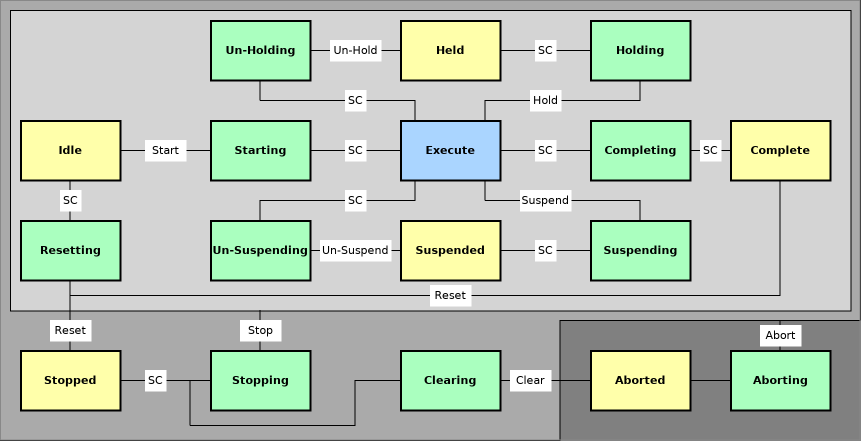
VISUALIZATION VFM_PackML  // 861x441
VAR_IN_OUT
	HMI : ST_PackMLBaseModule_HMI;
END_VAR
    Rectangle (560,320 301x121)
    Rectangle (10,10 841x301)
    Rectangle (590,350 101x61), "Aborted", colour toggle: HMI.Status.State = Tc3_PackML_V2.E_PMLState.ePMLState_Aborted
    Rectangle (400,350 101x61), "Clearing", colour toggle: HMI.Status.State = Tc3_PackML_V2.E_PMLState.ePMLState_Clearing
    Rectangle (210,350 101x61), "Stopping", colour toggle: HMI.Status.State = Tc3_PackML_V2.E_PMLState.ePMLState_Stopping
    Rectangle (20,350 101x61), "Stopped", colour toggle: HMI.Status.State = Tc3_PackML_V2.E_PMLState.ePMLState_Stopped
    Rectangle (20,220 101x61), "Resetting", colour toggle: HMI.Status.State = Tc3_PackML_V2.E_PMLState.ePMLState_Resetting
    Rectangle (20,120 101x61), "Idle", colour toggle: HMI.Status.State = Tc3_PackML_V2.E_PMLState.ePMLState_Idle
    Rectangle (210,120 101x61), "Starting", colour toggle: HMI.Status.State = Tc3_PackML_V2.E_PMLState.ePMLState_Starting
    Rectangle (400,120 101x61), "Execute", colour toggle: HMI.Status.State = Tc3_PackML_V2.E_PMLState.ePMLState_Execute
    Rectangle (590,20 101x61), "Holding", colour toggle: HMI.Status.State = Tc3_PackML_V2.E_PMLState.ePMLState_Holding
    Rectangle (400,20 101x61), "Held", colour toggle: HMI.Status.State = Tc3_PackML_V2.E_PMLState.ePMLState_Held
    Rectangle (210,20 101x61), "Un-Holding", colour toggle: HMI.Status.State = Tc3_PackML_V2.E_PMLState.ePMLState_Unholding
    Rectangle (590,220 101x61), "Suspending", colour toggle: HMI.Status.State = Tc3_PackML_V2.E_PMLState.ePMLState_Suspending
    Rectangle (400,220 101x61), "Suspended", colour toggle: HMI.Status.State = Tc3_PackML_V2.E_PMLState.ePMLState_Suspended
    Rectangle (210,220 101x61), "Un-Suspending", colour toggle: HMI.Status.State = Tc3_PackML_V2.E_PMLState.ePMLState_Unsuspending
    Rectangle (590,120 101x61), "Completing", colour toggle: HMI.Status.State = Tc3_PackML_V2.E_PMLState.ePMLState_Completing
    Rectangle (730,120 101x61), "Complete", colour toggle: HMI.Status.State = Tc3_PackML_V2.E_PMLState.ePMLState_Complete
    Rectangle (730,350 101x61), "Aborting", colour toggle: HMI.Status.State = Tc3_PackML_V2.E_PMLState.ePMLState_Aborting
    Line (0,0) (860,0)
    Line (860,0) (860,320)
    Line (560,320) (860,320)
    Line (560,440) (560,320)
    Line (0,440) (560,440)
    Line (0,440) (0,0)
    Line (780,350) (780,320)
    Line (690,380) (730,380)
    Line (355,380) (400,380)
    Line (500,380) (590,380)
    Line (355,425) (355,380)
    Line (190,425) (355,425)
    Line (260,350) (260,310)
    Line (120,380) (210,380)
    Line (310,250) (400,250)
    Line (500,250) (590,250)
    Line (500,50) (590,50)
    Line (310,50) (400,50)
    Line (120,150) (210,150)
    Line (310,150) (400,150)
    Line (500,150) (590,150)
    Line (690,150) (730,150)
    Line (70,295) (780,295)
    Line (190,425) (190,380)
    Line (70,350) (70,280)
    Line (780,295) (780,180)
    Line (70,220) (70,180)
    Line (485,100) (640,100)
    Line (640,100) (640,80)
    Line (485,120) (485,100)
    Line (640,220) (640,200)
    Line (485,200) (640,200)
    Line (485,200) (485,180)
    Line (260,100) (260,80)
    Line (415,120) (415,100)
    Line (260,100) (415,100)
    Line (260,220) (260,200)
    Line (260,200) (415,200)
    Line (415,200) (415,180)
    Rectangle (760,325 41x21), "Abort"
    Rectangle (50,320 41x21), "Reset"
    Rectangle (510,370 41x21), "Clear"
    Rectangle (240,320 41x21), "Stop"
    Rectangle (145,370 21x21), "SC"
    Rectangle (60,190 21x21), "SC"
    Rectangle (345,140 21x21), "SC"
    Rectangle (535,140 21x21), "SC"
    Rectangle (535,40 21x21), "SC"
    Rectangle (700,140 21x21), "SC"
    Rectangle (535,240 21x21), "SC"
    Rectangle (345,190 21x21), "SC"
    Rectangle (345,90 21x21), "SC"
    Rectangle (530,90 31x21), "Hold"
    Rectangle (520,190 51x21), "Suspend"
    Rectangle (320,240 71x21), "Un-Suspend"
    Rectangle (330,40 51x21), "Un-Hold"
    Rectangle (430,285 41x21), "Reset"
    Rectangle (145,140 41x21), "Start"
END_VISUALIZATION

(* stored: Version 1.1.0.1, ProductVersion 3.1.4024.12
   Visu VFM_PackML: Id {b7914f68-723c-465c-80d5-939c603d3086} *)
